FUNCTION_BLOCK AxisVelocityTestSuite EXTENDS TestSuite<TestSuiteParameter.MaxTestCount>
VAR
	StubAxis : AXIS_REF;
	iStubTask : I_Task;
	TestAxisHalt : VelocityBehaviour(StubAxis);
END_VAR

END_FUNCTION_BLOCK

(* stored: Version 1.1.0.1
   POU AxisVelocityTestSuite: Id {6f423009-7ac9-4bbc-9784-ede5e34ea635}, SpecialFunc None *)
